{attribute 'qualified_only'}
VAR_GLOBAL
	//Time
	stTime : ST_Time;
	bUPSDetect : BOOL;
END_VAR

VAR_GLOBAL PERSISTENT
	sUserLogged					:STRING;
	cntResettable				:FB_Counter;
	cntHourly					:FB_Counter;
	cntTotal					:FB_Counter;
	cntBatch					:FB_Counter;
	cntShift1					:FB_Counter;
	cntShift2					:FB_Counter;
	cntShift3					:FB_Counter;
	stSettings					:ST_Settings;
	aTrays						:ARRAY[1..10] OF ARRAY[1..14,1..7] OF BOOL;
END_VAR

(* stored: Version 1.1.0.1
   GVL GV: Id {07af1401-1339-48c1-8486-bb5ea9b2636f} *)
